TYPE st01 :
STRUCT
	r1:LREAL;
	i1:INT;
	s1:STRING;
	s2:STRING;
	r2:LREAL;
	i2:INT;
END_STRUCT
END_TYPE

(* stored: Version 1.1.0.1, ProductVersion 3.1.4024.12
   DUT st01: Id {fb4bd03f-17e4-4ac4-8df5-ae7909b99b32} *)
